TYPE (* A Structure with 4 Bits *)
  (* Version 1.0, 2024-02-21, franz *)
  st04b : STRUCT
    b00 : BOOL; (* BIT 00 *)
    b01 : BOOL; (* BIT 01 *)
    b02 : BOOL; (* BIT 02 *)
    b03 : BOOL; (* BIT 03 *)
  END_STRUCT;
END_TYPE
